// TIA Portal V16 export
// export: Created 2024-12-03T15:41:45.2028352Z, ExportSetting WithReadOnly, DisplayName Totally Integrated Automation Portal, DisplayVersion V16 Update 6, DisplayName TIA Portal Version Control Interface, DisplayVersion V16 Update 2, DisplayName TIA Portal Openness, DisplayVersion V16 Update 6, DisplayName TIA Portal Teamcenter Gateway, DisplayVersion V16, DisplayName SINAMICS Startdrive Advanced, DisplayVersion V16 Update 5, DisplayName SINAMICS Startdrive G130, G150, S120, S150, SINAMICS MV, S210, DisplayVersion V16 Update 5, DisplayName SINAMICS Startdrive G110M, G120, G120C, G120D, G120P, G115D, DisplayVersion V16 Update 5, DisplayName STEP 7 Professional, DisplayVersion V16 Update 6, DisplayName STEP 7 Safety, DisplayVersion V16, DisplayName WinCC Advanced / Unified PC, DisplayVersion V16 Update 6
TYPE "Q_Mettler_UDT"
// stored: CreationDate 2022-02-16T10:42:03.057947Z, InterfaceModifiedDate 2022-02-16T12:11:34.8048806Z, IsConsistent true, LibraryConformanceStatus The object is library-conformant., ModifiedDate 2022-02-16T12:11:34.8048806Z
   STRUCT
      CommandValue : Real;
      channelMask : Word;
      Command : Word;
   END_STRUCT;
END_TYPE
